{attribute 'qualified_only'}
VAR_GLOBAL
	bAuto 		: BOOL;
	
END_VAR

(* stored: Version 1.1.0.1, ProductVersion 3.1.4024.12
   GVL HMI: Id {4daaeb84-52ae-4b66-b477-32ed02fdace7} *)
